(* CODESYS project proj_11_15_zad1_z_uwagami.project

Project tree, tasks and I/O mapping:
  Device : Berghof MX6 Control, Berghof Automation GmbH, version 1.8.0.0
    application Application
      libraries: Standard, * (System)
      task MainTask (cyclic, interval t#25ms, priority 1) calls PLC_PRG
      program PLC_PRG [LD]
      visualisation Visualization
    Extension_Slots : Extension Slots, Berghof Automation GmbH, version 1.2.0.3
      XBIO_Berghof_IO : XBIO Berghof IO, Berghof Automation GmbH, version 1.2.0.3
          unmapped channels: Digital Input 0, Digital Input 1, Digital Input 2, Digital Input 3, Digital Input 4, Digital Output 0, Digital Output 1, Digital Output 2, Digital Output 3, Digital Output 4, Channel 0, Channel 1, Channel 2, Channel 3, Channel 4, Channel 5, Channel 6, Channel 7, Channel 8, Channel 9, Channel 10, Channel 11, Channel 0, Channel 1, Channel 2, Channel 3, Channel 4, Channel 5, Channel 6, Channel 7, Counter/Encoder 0, Counter/Encoder 1, Differential Counter/Encoder (0+1), DUMMY 0
      <Empty>
  text list GlobalTextList
*)

// Device/Application/PLC_PRG
PROGRAM PLC_PRG
VAR_OUTPUT
	Q3_CZERWONE_POJAZDY AT %QX0.2: BOOL;
	Q2_ZOLTE_POJAZDY AT %QX0.1: BOOL;
	Q1_ZIELONE_POJAZDY AT %QX0.0: BOOL;
	Q5_CZERWONE_PIESI AT %QX0.4: BOOL;
END_VAR
VAR
	S1: BOOL;
	S2: BOOL;
	S3: BOOL;
	TON2: TON;
	T1: TIME;
	TON1: TON;
	T2: TIME;
	CTU: CTU;
	CNT: WORD;
	M_MRUG1: BOOL;
	M2: BOOL;
	TON_8: TON;
	TONCTU: TON;
	TONCTU1: TON;
	CTD1: CTD;
	TONCTD1: TON;
	M3: BOOL;
	M4: BOOL;
	MSUB1: BOOL;
	MSUBCZ: BOOL;
	M5: BOOL;
	TONCTD2: TON;
	PTCTD2: TIME := T#0.5S;
	TCTD2: TIME;
	MSUBZ: BOOL;
	MLOADZ: BOOL;
	CZI: WORD;
	M6: BOOL;
	M7: BOOL;
	TONCTD3: TON;
	TONCTD4: TON;
	PTCTD3: TIME := T#0.5S;
	TCTD3: TIME;
	PTCTD4: TIME := T#0.5S;
	TCTD4: TIME;
	CTD2: CTD;
END_VAR
VAR_OUTPUT
	Q4_ZIELONE_PIESI AT %QX0.3: BOOL;
	Q6_KONTROLKA AT %QX0.5: BOOL;
END_VAR
VAR
	X1_TRYB: BOOL;
	X2_PRZYCISK: BOOL;
	S0: BOOL;
	S4: BOOL;
	S5: BOOL;
	S6: BOOL;
	TON0: TON;
	TON3: TON;
	TON4: TON;
	TON5: TON;
	TON6: TON;
	T0: TIME;
	T3: TIME;
	T4: TIME;
	T5: TIME;
	T6: TIME;
	TON_MRUG0: TON;
	TON_MRUG1: TON;
	T_MRUG0: TIME;
	T_MRUG1: TIME;
	M_MRUG0: BOOL;
	M_MRUG2: BOOL;
	S1_SET: BOOL;
	TON7: TON;
	T7: TIME;
	X3_REQUEST: BOOL;
	S_P: BOOL;
	M_MRUG3: BOOL;
	TON_MRUG2: TON;
	TON_MRUG3: TON;
	T_MRUG2: TIME;
	T_MRUG3: TIME;
	PT0: TIME := T#3S;
	PT1: TIME := T#2S;
	PT2: TIME := T#5S;
	PT3: TIME := T#3S;
	PT4: TIME := T#15S;
	PT5: TIME := T#6S;
	PT6: TIME := T#3S;
	PT7: TIME := T#3S;
	PTCZ: TIME;
	PTZ1: TIME;
	PTZ: TIME;
	M1: BOOL;
	PZI: WORD;
	PCZI: WORD;
	PTCTD1: TIME := T#0.5S;
	TCTD1: TIME;
	CCZ: WORD;
END_VAR
VAR // added by the converter: edge detectors and wires of the graphical bodies
    _w1, _w2, _w3, _w4, _w5, _w6 : BOOL;
END_VAR

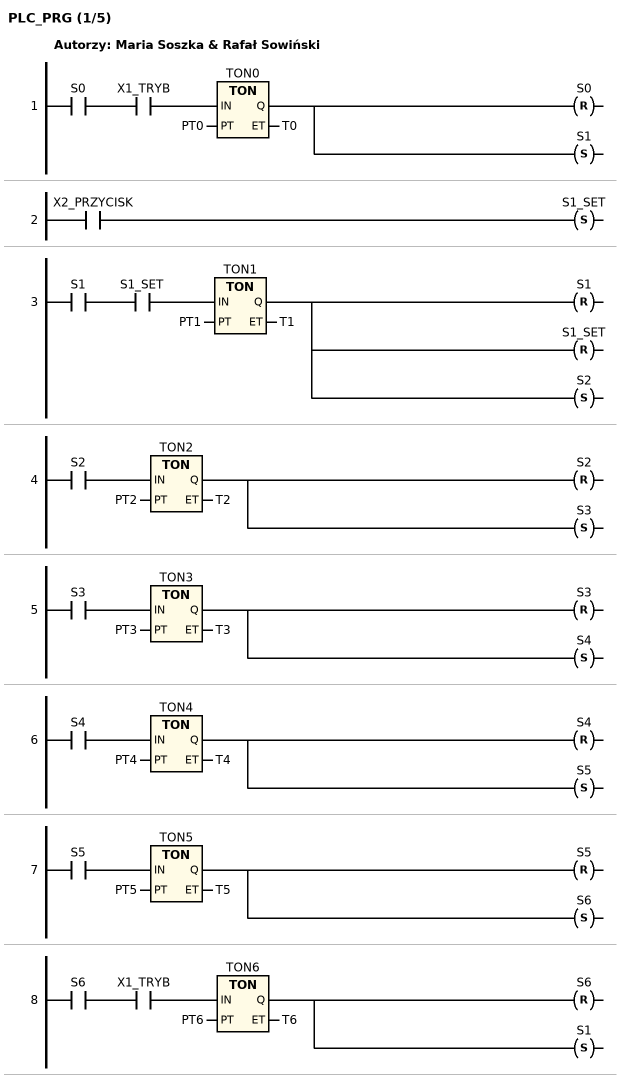
// NETWORK 1: Autorzy: Maria Soszka & Rafał Sowiński
TON0(IN := S0 AND X1_TRYB, PT := PT0, ET => T0); // TON
S0 R= TON0.Q;
S1 S= TON0.Q;

// NETWORK 2
S1_SET S= X2_PRZYCISK;

// NETWORK 3
TON1(IN := S1 AND S1_SET, PT := PT1, ET => T1); // TON
S1 R= TON1.Q;
S1_SET R= TON1.Q;
S2 S= TON1.Q;

// NETWORK 4
TON2(IN := S2, PT := PT2, ET => T2); // TON
S2 R= TON2.Q;
S3 S= TON2.Q;

// NETWORK 5
TON3(IN := S3, PT := PT3, ET => T3); // TON
S3 R= TON3.Q;
S4 S= TON3.Q;

// NETWORK 6
TON4(IN := S4, PT := PT4, ET => T4); // TON
S4 R= TON4.Q;
S5 S= TON4.Q;

// NETWORK 7
TON5(IN := S5, PT := PT5, ET => T5); // TON
S5 R= TON5.Q;
S6 S= TON5.Q;

// NETWORK 8
TON6(IN := S6 AND X1_TRYB, PT := PT6, ET => T6); // TON
S6 R= TON6.Q;
S1 S= TON6.Q;

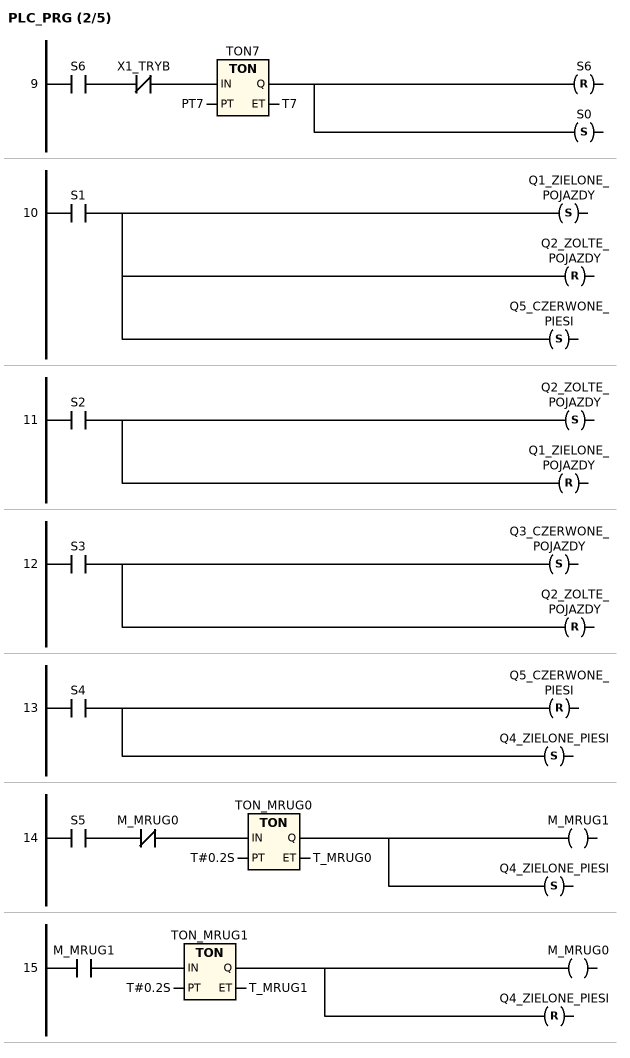
// NETWORK 9
TON7(IN := S6 AND NOT X1_TRYB, PT := PT7, ET => T7); // TON
S6 R= TON7.Q;
S0 S= TON7.Q;

// NETWORK 10
Q1_ZIELONE_POJAZDY S= S1;
Q2_ZOLTE_POJAZDY R= S1;
Q5_CZERWONE_PIESI S= S1;

// NETWORK 11
Q2_ZOLTE_POJAZDY S= S2;
Q1_ZIELONE_POJAZDY R= S2;

// NETWORK 12
Q3_CZERWONE_POJAZDY S= S3;
Q2_ZOLTE_POJAZDY R= S3;

// NETWORK 13
Q5_CZERWONE_PIESI R= S4;
Q4_ZIELONE_PIESI S= S4;

// NETWORK 14
TON_MRUG0(IN := S5 AND NOT M_MRUG0, PT := T#0.2S, ET => T_MRUG0); // TON
M_MRUG1 := TON_MRUG0.Q;
Q4_ZIELONE_PIESI S= TON_MRUG0.Q;

// NETWORK 15
TON_MRUG1(IN := M_MRUG1, PT := T#0.2S, ET => T_MRUG1); // TON
M_MRUG0 := TON_MRUG1.Q;
Q4_ZIELONE_PIESI R= TON_MRUG1.Q;

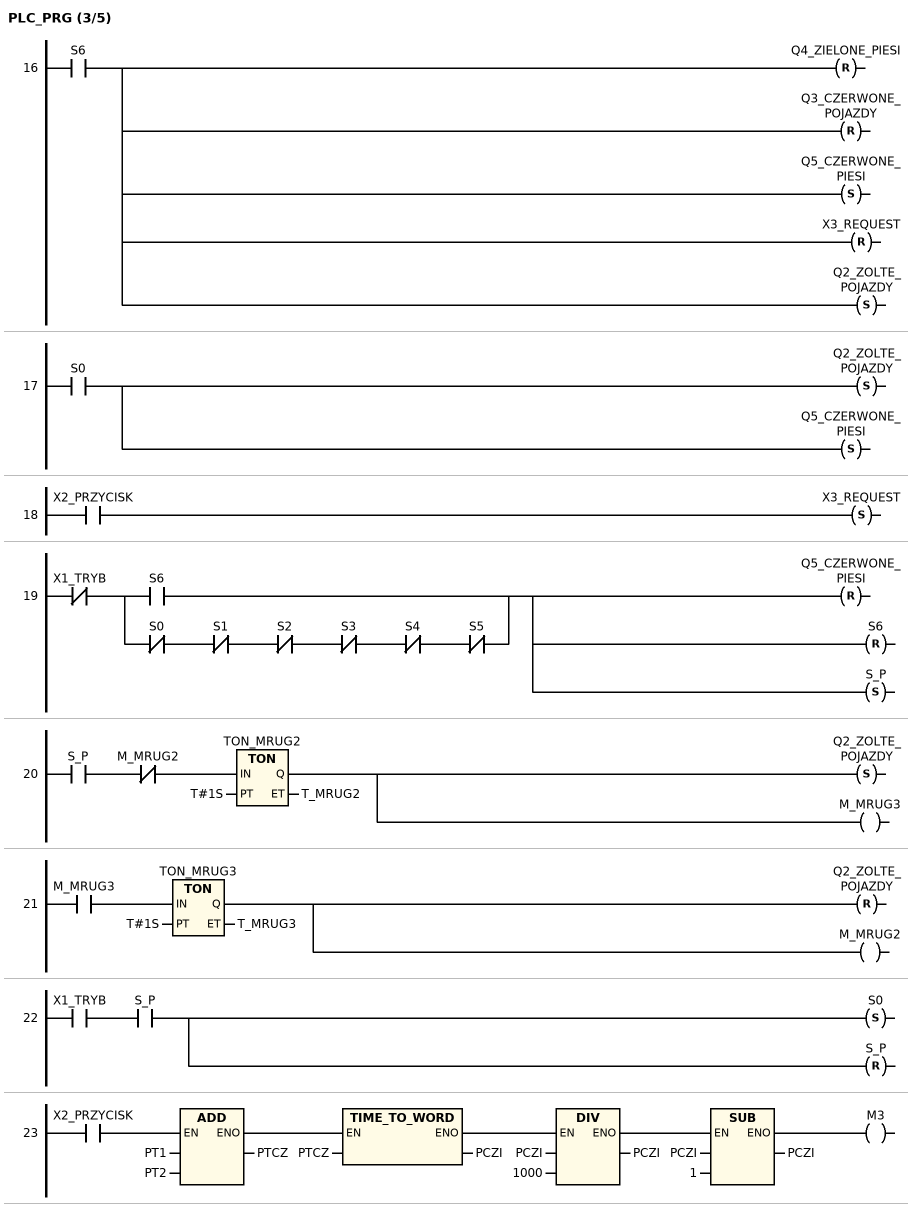
// NETWORK 16
Q4_ZIELONE_PIESI R= S6;
Q3_CZERWONE_POJAZDY R= S6;
Q5_CZERWONE_PIESI S= S6;
X3_REQUEST R= S6;
Q2_ZOLTE_POJAZDY S= S6;

// NETWORK 17
Q2_ZOLTE_POJAZDY S= S0;
Q5_CZERWONE_PIESI S= S0;

// NETWORK 18
X3_REQUEST S= X2_PRZYCISK;

// NETWORK 19
_w1 := NOT X1_TRYB AND (S6 OR NOT S0 AND NOT S1 AND NOT S2 AND NOT S3 AND NOT S4 AND NOT S5);
Q5_CZERWONE_PIESI R= _w1;
S6 R= _w1;
S_P S= _w1;

// NETWORK 20
TON_MRUG2(IN := S_P AND NOT M_MRUG2, PT := T#1S, ET => T_MRUG2); // TON
Q2_ZOLTE_POJAZDY S= TON_MRUG2.Q;
M_MRUG3 := TON_MRUG2.Q;

// NETWORK 21
TON_MRUG3(IN := M_MRUG3, PT := T#1S, ET => T_MRUG3); // TON
Q2_ZOLTE_POJAZDY R= TON_MRUG3.Q;
M_MRUG2 := TON_MRUG3.Q;

// NETWORK 22
_w2 := X1_TRYB AND S_P;
S0 S= _w2;
S_P R= _w2;

// NETWORK 23
_w3 := X2_PRZYCISK;
IF _w3 THEN PTCZ := PT1 + PT2; END_IF
IF _w3 THEN PCZI := TIME_TO_WORD(PTCZ); END_IF
IF _w3 THEN PCZI := PCZI / 1000; END_IF
IF _w3 THEN PCZI := PCZI - 1; END_IF
M3 := _w3;

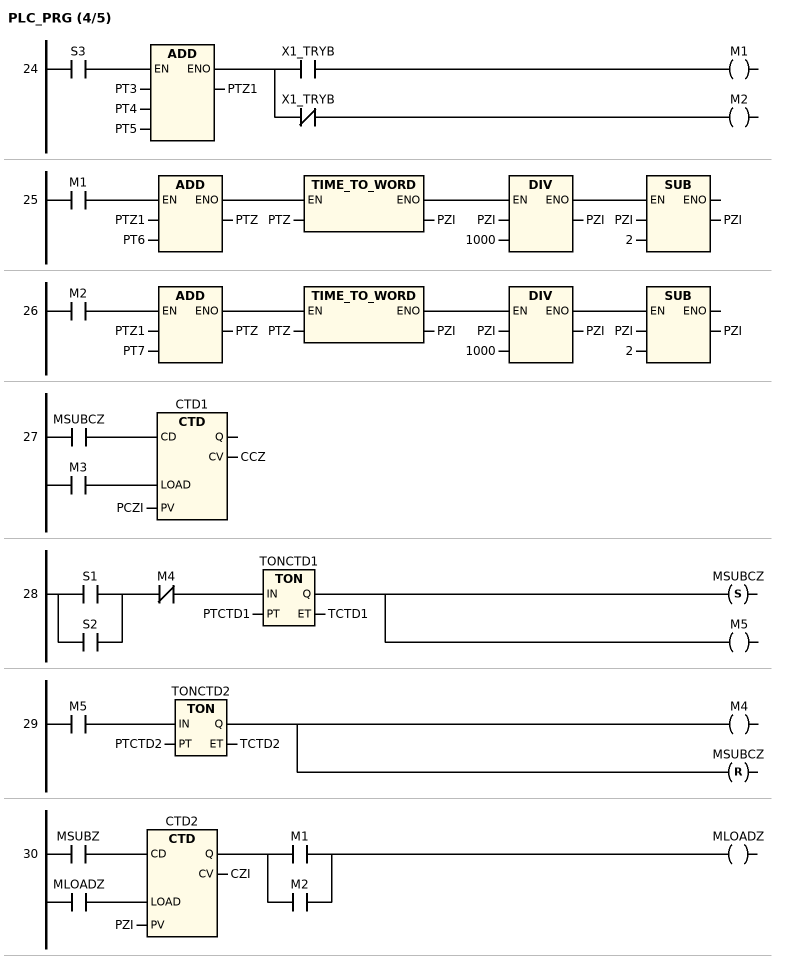
// NETWORK 24
_w4 := S3;
IF _w4 THEN PTZ1 := PT3 + PT4 + PT5; END_IF
M1 := _w4 AND X1_TRYB;
M2 := _w4 AND NOT X1_TRYB;

// NETWORK 25
_w5 := M1;
IF _w5 THEN PTZ := PTZ1 + PT6; END_IF
IF _w5 THEN PZI := TIME_TO_WORD(PTZ); END_IF
IF _w5 THEN PZI := PZI / 1000; END_IF
IF _w5 THEN PZI := PZI - 2; END_IF

// NETWORK 26
_w6 := M2;
IF _w6 THEN PTZ := PTZ1 + PT7; END_IF
IF _w6 THEN PZI := TIME_TO_WORD(PTZ); END_IF
IF _w6 THEN PZI := PZI / 1000; END_IF
IF _w6 THEN PZI := PZI - 2; END_IF

// NETWORK 27
CTD1(CD := MSUBCZ, LOAD := M3, PV := PCZI, CV => CCZ); // CTD

// NETWORK 28
TONCTD1(IN := (S1 OR S2) AND NOT M4, PT := PTCTD1, ET => TCTD1); // TON
MSUBCZ S= TONCTD1.Q;
M5 := TONCTD1.Q;

// NETWORK 29
TONCTD2(IN := M5, PT := PTCTD2, ET => TCTD2); // TON
M4 := TONCTD2.Q;
MSUBCZ R= TONCTD2.Q;

// NETWORK 30
CTD2(CD := MSUBZ, LOAD := MLOADZ, PV := PZI, CV => CZI); // CTD
MLOADZ := CTD2.Q AND (M1 OR M2);

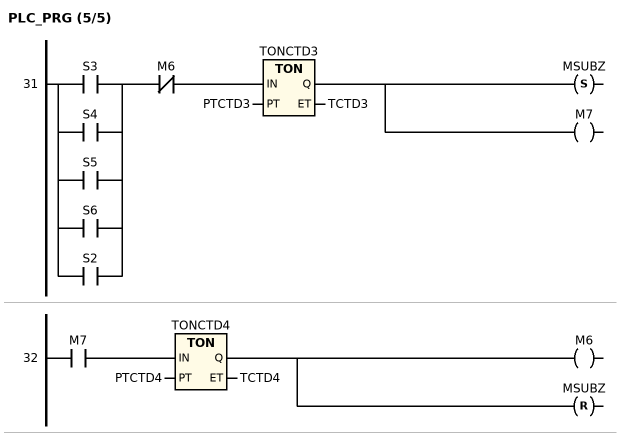
// NETWORK 31
TONCTD3(IN := (S3 OR S4 OR S5 OR S6 OR S2) AND NOT M6, PT := PTCTD3, ET => TCTD3); // TON
MSUBZ S= TONCTD3.Q;
M7 := TONCTD3.Q;

// NETWORK 32
TONCTD4(IN := M7, PT := PTCTD4, ET => TCTD4); // TON
M6 := TONCTD4.Q;
MSUBZ R= TONCTD4.Q;

END_PROGRAM

// Device/Application/Visualization
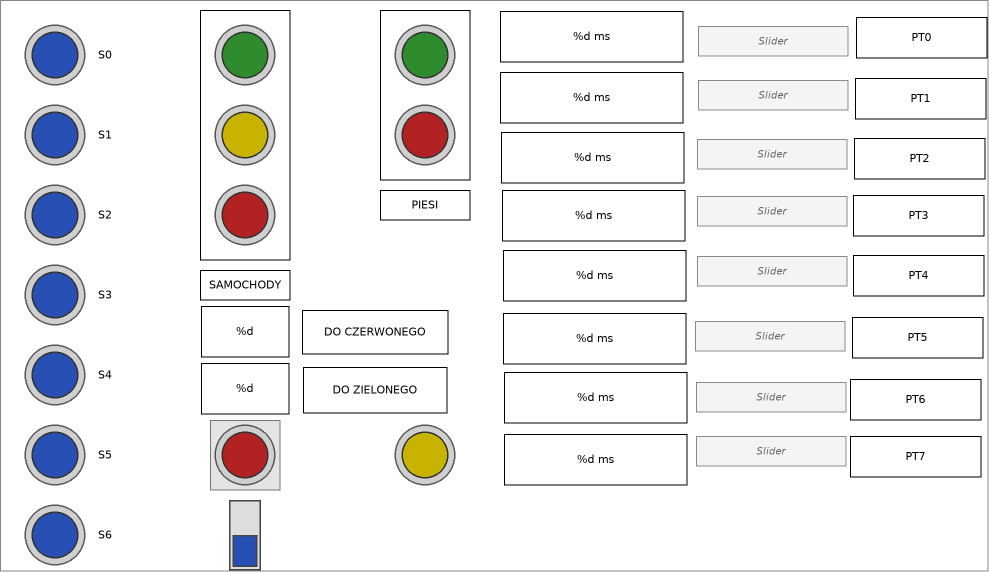
VISUALIZATION Visualization  // 989x572
    Rectangle (380,190 90x30)
    Rectangle (380,10 90x170)
    Rectangle (200,10 90x250)
    Lamp1 (210,20 70x70), variable: PLC_PRG.Q1_ZIELONE_POJAZDY, style: Lamp-Lamp1-Green
    Lamp1 (210,100 70x70), variable: PLC_PRG.Q2_ZOLTE_POJAZDY, style: Lamp-Lamp1-Yellow
    Lamp1 (210,180 70x70), variable: PLC_PRG.Q3_CZERWONE_POJAZDY, style: Lamp-Lamp1-Red
    Lamp1 (390,20 70x70), variable: PLC_PRG.Q4_ZIELONE_PIESI, style: Lamp-Lamp1-Green
    Lamp1 (390,100 70x70), variable: PLC_PRG.Q5_CZERWONE_PIESI, style: Lamp-Lamp1-Red
    Lamp1 (20,20 70x70), variable: PLC_PRG.S0, style: Lamp-Lamp1-Blue
    Lamp1 (20,100 70x70), variable: PLC_PRG.S1, style: Lamp-Lamp1-Blue
    Lamp1 (20,180 70x70), variable: PLC_PRG.S2, style: Lamp-Lamp1-Blue
    Lamp1 (20,260 70x70), variable: PLC_PRG.S3, style: Lamp-Lamp1-Blue
    Lamp1 (20,340 70x70), variable: PLC_PRG.S4, style: Lamp-Lamp1-Blue
    Lamp1 (20,420 70x70), variable: PLC_PRG.S5, style: Lamp-Lamp1-Blue
    Lamp1 (20,500 70x70), variable: PLC_PRG.S6, style: Lamp-Lamp1-Blue
    DipSwitch (210,500 70x70), variable: PLC_PRG.X1_TRYB, behaviour: TOGGLE, style: Switch-DipSwitch-Blue
    PushSwitch (210,420 70x70), variable: PLC_PRG.X2_PRZYCISK, behaviour: TAP, style: Switch-PushSwitch-Red
    Label (390,190 70x30), "PIESI"
    Rectangle (200,270 90x30)
    Label (200,250 90x70), "SAMOCHODY"
    Label (30,280 150x30), "S3"
    Label (30,40 150x30), "S0"
    Label (30,200 150x30), "S2"
    Label (30,120 150x30), "S1"
    Label (30,360 150x30), "S4"
    Label (30,440 150x30), "S5"
    Label (30,520 150x30), "S6"
    Lamp1 (390,420 70x70), variable: PLC_PRG.X3_REQUEST, style: Lamp-Lamp1-Yellow
    Rectangle (500,11 183x51), "%d ms", text variable: PLC_PRG.PT0
    Rectangle (500,72 183x51), "%d ms", text variable: PLC_PRG.PT1
    Rectangle (501,132 183x51), "%d ms", text variable: PLC_PRG.PT2
    Rectangle (502,190 183x51), "%d ms", text variable: PLC_PRG.PT3
    Rectangle (503,250 183x51), "%d ms", text variable: PLC_PRG.PT4
    Rectangle (503,313 183x51), "%d ms", text variable: PLC_PRG.PT5
    Rectangle (504,372 183x51), "%d ms", text variable: PLC_PRG.PT6
    Rectangle (504,434 183x51), "%d ms", text variable: PLC_PRG.PT7
    Slider (698,26 150x30), variable: PLC_PRG.PT0, scale 100..20000
    Slider (698,80 150x30), variable: PLC_PRG.PT1, scale 100..20000
    Slider (697,139 150x30), variable: PLC_PRG.PT2, scale 100..20000
    Slider (697,196 150x30), variable: PLC_PRG.PT3, scale 100..20000
    Slider (697,256 150x30), variable: PLC_PRG.PT4, scale 100..20000
    Slider (695,321 150x30), variable: PLC_PRG.PT5, scale 100..20000
    Slider (696,382 150x30), variable: PLC_PRG.PT6, scale 100..20000
    Slider (696,436 150x30), variable: PLC_PRG.PT7, scale 100..20000
    Rectangle (856,17 131x41), "PT0"
    Rectangle (855,78 131x41), "PT1"
    Rectangle (854,138 131x41), "PT2"
    Rectangle (853,195 131x41), "PT3"
    Rectangle (853,255 131x41), "PT4"
    Rectangle (852,317 131x41), "PT5"
    Rectangle (850,379 131x41), "PT6"
    Rectangle (850,436 131x41), "PT7"
    Rectangle (201,306 88x51), "%d", text variable: PLC_PRG.CCZ
    Rectangle (201,363 88x51), "%d", text variable: PLC_PRG.CZI
    Rectangle (302,310 146x44), "DO CZERWONEGO"
    Rectangle (303,367 144x46), "DO ZIELONEGO"
END_VISUALIZATION
